(* PLC project CoDeSys External Library Template, WAGO e!COCKPIT e!COCKPIT, author 3S - Smart Software Solutions GmbH *)
(* stored: creationDateTime 2019-10-29T12:37:19.3718897, version 3.5.5.30, modificationDateTime 2019-10-29T12:36:39.3744516, organization 3S - Smart Software Solutions GmbH *)
(* Library project template with all possible element types, docu and a sample project structure *)

(* values of enumPPPSHarmonogramy: Ekonomiczny: Tryb pracy ekonomicznej; Komfort: Tryb pracy komfortu *)

(* Autor: Paweł Kąkol, 2018-09-10-PK Prawa majątkowe: Solwena Sp. z o.o., Aktualizacje: Opis: enum służy do obsługi Trybów pracy harmonogramu na budynkach PPP Sopot (ENGIE) *)
{attribute 'qualified_only'}
{attribute 'strict'}
TYPE enumPPPSHarmonogramy : (Ekonomiczny := 0, Komfort := 1);
END_TYPE
